{attribute 'qualified_only'}
VAR_GLOBAL
END_VAR

(* stored: Version 1.1.0.1, ProductVersion 3.1.4024.12
   GVL gvlIO: Id {b502dacf-f837-4a1a-9176-5415efc890a4} *)
